Universal Robots PolyScope program: PythonSubprogram1a.urp

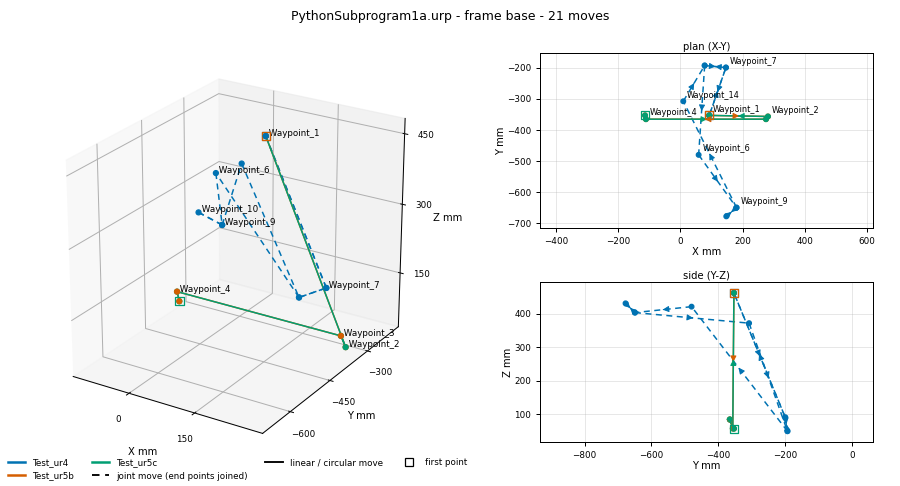
[picture p0: tool path of PythonSubprogram1a.urp in frame base, 21 of 21 moves have a stored position in this frame; points joined in program order, loops and branches not executed]
Program PythonSubprogram1a (installation=default directory=/programs/usbdisk/NoodleBotSoftware createdIn=3.12.1.90940 lastSavedIn=3.12.1.90940 robotSerialNumber=2017354841)
Calibrated DH parameters: a=[0.000094, -0.006117, -0.382762, 0.000086, 0.000044, 0]; d=[0.089236, 217.751846, -204.357806, -13.283746, 0.094902, 0.082641]; alpha=[1.57017, 0.001953, -0.006493, 1.570192, -1.570543, 0]; deltaTheta=[0.000036, 1.556386, -1.779789, 0.223359, -0.000014, -0.000001]
BeforeStart
  var_1 := socket_open("192.168.0.100",30000)
Robot Program (runOnlyOnce=false)
  Loop While (checkContinuously=false) expression=var_1≟ False
    var_1 := socket_open("192.168.0.100",30000)
    Wait Sleep waitTime=0.5
  Script: socket_send_string("asking_for_data")
  Wait Sleep waitTime=0.5
  var_2 := socket_read_ascii_float(3)
  Wait Sleep waitTime=0.5
  var_1 := False
  If var_2[1]≟1
    Call Test_ur4
  If var_2[1]≟1
    Call Test_ur5b
  If var_2[2]≟1 and digital_in[0]≟ False
    Set DigitalOutput pin=digital_out[4]; digitalValue=1
    Wait Sleep waitTime=3
    Set DigitalOutput pin=digital_out[4]; digitalValue=0
    Wait Sleep waitTime=0.5
    Set DigitalOutput pin=digital_out[5]; digitalValue=1
    Wait Sleep waitTime=3
    Set DigitalOutput pin=digital_out[5]; digitalValue=0
    Wait Sleep waitTime=0.5
  If var_2[3]≟1 and digital_in[0]≟ False
    Set DigitalOutput pin=digital_out[6]; digitalValue=1
    Wait Sleep waitTime=0.5
    Set DigitalOutput pin=digital_out[6]; digitalValue=0
    Wait Sleep waitTime=0.5
    Set DigitalOutput pin=digital_out[6]; digitalValue=1
    Wait Sleep waitTime=0.5
    Set DigitalOutput pin=digital_out[6]; digitalValue=0
    Wait Sleep waitTime=0.5
  If digital_in[0]≟ False
    Call Test_ur5c
    Wait Sleep waitTime=0.5
    var_1 := False
  Script: socket_close()
SubProgram -> Test_ur4
SubProgram -> Test_ur5c
SubProgram -> Test_ur5b
SubProgram Test_ur4 (keepSynchronizedWithDisk=false) programFile=/programs/Test ur4.urp
  MoveJ speed 120 deg/s, acceleration 90 deg/s^2 (useActiveTCP=true)
    URCap RG2 (RG - On Robot, OnRobot A/S) dataModel(depthCompensate=false, force=40, payload=0.0, width=50, name=RG2(50))
    Waypoint Waypoint_1: TCP in base x=92.939 y=-353.097 z=462.595 mm, rx=1.1692 ry=-1.2408 rz=1.1709 rad; joints [88.542, -137.018, 138.65, 178.588, 268.341, 89.999] deg; flange x=103.097 y=-166.778 z=463.297 mm, rx=1.2543 ry=1.1818 rz=-1.2438 rad
    Wait Sleep waitTime=1
    Waypoint Waypoint_7: TCP in base x=146.59 y=-199.362 z=90.11 mm, rx=-2.576 ry=0.0709 rz=1.786 rad; joints [138.196, -78.978, 116.17, 296.94, 232.836, 75.177] deg; flange x=321.213 y=-205.121 z=155.617 mm, rx=-0.0531 ry=-1.9288 rz=-0.0072 rad
    Waypoint Waypoint_8: motionParameters(jointSpeed=1.047198 jointAcceleration=1.396263 cartesianSpeed=0.25 cartesianAcceleration=1.2); TCP in base x=78.27 y=-192.88 z=48.88 mm, rx=2.2302 ry=-0.0356 rz=-2.1945 rad; joints [134.566, -66.419, 124.008, 301.345, 224.751, 90.836] deg; flange x=264.839 y=-194.194 z=51.908 mm, rx=-0.0253 ry=-1.5868 rz=0.0141 rad
    URCap RG2 (RG - On Robot, OnRobot A/S) dataModel(depthCompensate=false, force=40, payload=0.0, width=0, name=RG2(0))
    Waypoint Waypoint_6: motionParameters(jointSpeed=3.141593 jointAcceleration=4.363323 cartesianSpeed=0.25 cartesianAcceleration=1.2); TCP in base x=58.909 y=-479.811 z=421.549 mm, rx=1.7821 ry=-0.1873 rz=-1.5062 rad; joints [116.062, -88.461, 90.35, 328.087, 178.647, 99.309] deg; flange x=224.655 y=-394.146 z=420.424 mm, rx=-0.1714 ry=-1.6303 rz=0.9063 rad
    Waypoint Waypoint_9: motionParameters(jointSpeed=3.141593 jointAcceleration=7.853982 cartesianSpeed=0.25 cartesianAcceleration=1.2); TCP in base x=180.596 y=-649.229 z=403.821 mm, rx=1.6144 ry=0.2541 rz=-1.3829 rad; joints [117.26, -70.546, 74.017, 340.205, 157.34, 106.049] deg; flange x=301.868 y=-508.767 z=384.579 mm, rx=0.2448 ry=-1.5551 rz=1.1276 rad
    Waypoint Waypoint_10: motionParameters(jointSpeed=3.141593 jointAcceleration=11.34464 cartesianSpeed=0.25 cartesianAcceleration=1.2); TCP in base x=147.694 y=-677.333 z=431.472 mm, rx=0.6942 ry=-1.3705 rz=0.0188 rad; joints [115.407, -61.812, 59.106, 312.808, 176.983, 193.94] deg; flange x=313.081 y=-591.119 z=424.997 mm, rx=1.9367 ry=0.981 rz=-2.2472 rad
    Wait Sleep waitTime=0.5
    Waypoint Waypoint_11: motionParameters(jointSpeed=3.141593 jointAcceleration=26.179939 cartesianSpeed=0.25 cartesianAcceleration=1.2); TCP in base x=180.596 y=-649.229 z=403.821 mm, rx=1.6144 ry=0.2541 rz=-1.3829 rad; joints [117.26, -70.546, 74.017, 340.205, 157.34, 106.049] deg; flange x=301.868 y=-508.767 z=384.579 mm, rx=0.2448 ry=-1.5551 rz=1.1276 rad
    Set DigitalOutput pin=digital_out[7]; digitalValue=1
    Waypoint Waypoint_14: TCP in base x=9.564 y=-307.679 z=372.171 mm, rx=2.0617 ry=-0.361 rz=-1.9317 rad; joints [117.287, -91.513, 96.391, 348.159, 205.139, 106.043] deg; flange x=195.694 y=-300.018 z=382.774 mm, rx=-0.2824 ry=-1.6133 rz=0.3293 rad
    Waypoint Waypoint_12: TCP in base x=78.27 y=-192.88 z=48.88 mm, rx=2.2302 ry=-0.0356 rz=-2.1945 rad; joints [134.566, -66.419, 124.008, 301.345, 224.751, 90.836] deg; flange x=264.839 y=-194.194 z=51.908 mm, rx=-0.0253 ry=-1.5868 rz=0.0141 rad
    URCap RG2 (RG - On Robot, OnRobot A/S) dataModel(depthCompensate=false, force=40, payload=0.0, width=50, name=RG2(50))
    Waypoint Waypoint_13: TCP in base x=146.59 y=-199.362 z=90.11 mm, rx=-2.576 ry=0.0709 rz=1.786 rad; joints [138.196, -78.978, 116.17, 296.94, 232.836, 75.177] deg; flange x=321.213 y=-205.121 z=155.617 mm, rx=-0.0531 ry=-1.9288 rz=-0.0072 rad
    Wait Sleep waitTime=1
    Waypoint Waypoint_1: TCP in base x=92.939 y=-353.097 z=462.595 mm, rx=1.1692 ry=-1.2408 rz=1.1709 rad; joints [88.542, -137.018, 138.65, 178.588, 268.341, 89.999] deg; flange x=103.097 y=-166.778 z=463.297 mm, rx=1.2543 ry=1.1818 rz=-1.2438 rad
    Set DigitalOutput pin=digital_out[7]; digitalValue=0
SubProgram Test_ur5b (keepSynchronizedWithDisk=false) programFile=/programs/Test ur5b.urp
  MoveL speed 1000 mm/s, acceleration 1200 mm/s^2 (useActiveTCP=true) feature=Base
    URCap RG2 (RG - On Robot, OnRobot A/S) dataModel(depthCompensate=false, force=40, payload=0.0, width=85, name=RG2(85))
    Waypoint Waypoint_1: TCP in base x=92.939 y=-353.097 z=462.595 mm, rx=1.1692 ry=-1.2408 rz=1.1709 rad; joints [88.542, -137.018, 138.65, 178.588, 268.341, 89.999] deg; flange x=103.097 y=-166.778 z=463.297 mm, rx=1.2543 ry=1.1818 rz=-1.2438 rad
    Wait Sleep waitTime=0.1
    Waypoint Waypoint_2: TCP in base x=281.568 y=-356.493 z=57.062 mm, rx=2.4509 ry=-1.0812 rz=-0.3973 rad; joints [131.142, -83.255, 116.241, 241.937, 240.139, 90.003] deg; flange x=360.116 y=-306.414 z=218.729 mm, rx=-1.1245 ry=-2.5488 rz=0.6202 rad
    URCap RG2 (RG - On Robot, OnRobot A/S) dataModel(depthCompensate=false, payload=0.0, force=40, width=0, name=RG2(0))
    Wait Sleep waitTime=0.1
    Waypoint Waypoint_3: TCP in base x=275.23 y=-365.244 z=83.858 mm, rx=2.4082 ry=-1.0628 rz=-0.4074 rad; joints [131.131, -84.8, 114.576, 244.685, 237.533, 90.016] deg; flange x=358.189 y=-309.185 z=241.34 mm, rx=-1.1149 ry=-2.5256 rz=0.6807 rad
    Wait Sleep waitTime=0.1
    Waypoint Waypoint_4: TCP in base x=-110.35 y=-365.263 z=83.889 mm, rx=2.4083 ry=-1.0627 rz=-0.4074 rad; joints [69.173, -109.993, 144.496, 207.947, 251.859, 22.112] deg; flange x=-27.414 y=-309.154 z=241.302 mm, rx=-1.1146 ry=-2.5256 rz=0.6805 rad
    Wait Sleep waitTime=0.1
    Waypoint Waypoint_5: TCP in base x=-113.251 y=-352.97 z=56.401 mm, rx=2.4743 ry=-1.0833 rz=-0.4569 rad; joints [69.146, -107.002, 145.454, 208.35, 250.31, 22.145] deg; flange x=-30.387 y=-310.642 z=218.159 mm, rx=-1.1049 ry=-2.5237 rz=0.5697 rad
    Wait Sleep waitTime=0.1
SubProgram Test_ur5c (keepSynchronizedWithDisk=false) programFile=/programs/Test ur5c.urp
  MoveL speed 1000 mm/s, acceleration 1200 mm/s^2 (useActiveTCP=true) feature=Base
    Waypoint Waypoint_5: TCP in base x=-113.251 y=-352.97 z=56.401 mm, rx=2.4743 ry=-1.0833 rz=-0.4569 rad; joints [69.146, -107.002, 145.454, 208.35, 250.31, 22.145] deg; flange x=-30.387 y=-310.642 z=218.159 mm, rx=-1.1049 ry=-2.5237 rz=0.5697 rad
    Wait Sleep waitTime=0.1
    Waypoint Waypoint_4: TCP in base x=-110.35 y=-365.263 z=83.889 mm, rx=2.4083 ry=-1.0627 rz=-0.4074 rad; joints [69.173, -109.993, 144.496, 207.947, 251.859, 22.112] deg; flange x=-27.414 y=-309.154 z=241.302 mm, rx=-1.1146 ry=-2.5256 rz=0.6805 rad
    Wait Sleep waitTime=0.1
    Waypoint Waypoint_3: TCP in base x=275.23 y=-365.244 z=83.858 mm, rx=2.4082 ry=-1.0628 rz=-0.4074 rad; joints [131.131, -84.8, 114.576, 244.685, 237.533, 90.016] deg; flange x=358.189 y=-309.185 z=241.34 mm, rx=-1.1149 ry=-2.5256 rz=0.6807 rad
    Wait Sleep waitTime=0.1
    Waypoint Waypoint_2: TCP in base x=281.568 y=-356.493 z=57.062 mm, rx=2.4509 ry=-1.0812 rz=-0.3973 rad; joints [131.142, -83.255, 116.241, 241.937, 240.139, 90.003] deg; flange x=360.116 y=-306.414 z=218.729 mm, rx=-1.1245 ry=-2.5488 rz=0.6202 rad
    URCap RG2 (RG - On Robot, OnRobot A/S) dataModel(depthCompensate=false, force=40, payload=0.0, width=85, name=RG2(85))
    Wait Sleep waitTime=0.1
    Waypoint Waypoint_1: TCP in base x=92.939 y=-353.097 z=462.595 mm, rx=1.1692 ry=-1.2408 rz=1.1709 rad; joints [88.542, -137.018, 138.65, 178.588, 268.341, 89.999] deg; flange x=103.097 y=-166.778 z=463.297 mm, rx=1.2543 ry=1.1818 rz=-1.2438 rad
    Wait Sleep waitTime=0.1
    Set DigitalOutput pin=digital_out[7]; digitalValue=1
    Wait Sleep waitTime=7
    Set DigitalOutput pin=digital_out[7]; digitalValue=0
